// TIA Portal V20 export
DATA_BLOCK "EventsData"   // DB255
// stored: Access Published, MemoryReserve 100, Namespace Unit1
   VAR
      ResourceData { ExternalAccessible := 'False'; ExternalVisible := 'False'; ExternalWritable := 'False'} : "LPFE_typeResourceData";
      ValueEvent { ExternalAccessible := 'False'; ExternalVisible := 'False'; ExternalWritable := 'False'} : Struct
         EventDesctiption : WString[58];
         currentShift : USInt := 2;
         valueType : SInt := 11;
         productionCounter : DInt := 0;
      END_STRUCT;
      TelemetryContent : Array[0..20] of "LPFE_typeTelemetryContent";
      Taping : "LPFE_typeFlexNetData_10004";
      HeatPressLeft : "LPFE_typeFlexNetData_10004";
      HeatPressRight : "LPFE_typeFlexNetData_10004";
      HipotandThickness : "LPFE_typeFlexNetData_10004";
      Vision : "LPFE_typeFlexNetData_10004";
      Laser : "LPFE_typeFlexNetData_10004";
      Weight : "LPFE_typeFlexNetData_10004";
      RecordGenericPayload { S7_SetPoint := 'True'} : "LPFE_typeRecordGenericPayload";
   END_VAR
BEGIN
   ResourceData.resourceInterestID := 10;
END_DATA_BLOCK
